ADAPTER ISludgeHoldingTankStatus (* Adapter Interface *)
  (* Standard: 61499-1 *)
  (* Version 0.0, 24/08/2026, Schneider Electric *)
  PACKAGE SE.Nereda;
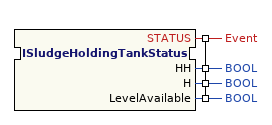
  EVENT_OUTPUT
    STATUS WITH HH, H, LevelAvailable;
  END_EVENT
  VAR_OUTPUT
    HH : BOOL; (* Confirmation Data from Plug *)
    H : BOOL; (* Indication Data from Plug *)
    LevelAvailable : BOOL;
  END_VAR
  SERVICE SOCKET/PLUG
    SEQUENCE request_confirm
      SOCKET.REQ(REQD) -> PLUG.REQ(REQD);
      PLUG.CNF(HH) -> SOCKET.CNF(HH);
    END_SEQUENCE
    SEQUENCE indication_response
      PLUG.IND(H) -> SOCKET.IND(H);
      SOCKET.RSP(RSPD) -> PLUG.RSP(RSPD);
    END_SEQUENCE
  END_SERVICE
END_ADAPTER
